(* PLC project Cell Example , CTH FIX1 1.0, author CTH SS2 *)
(* stored: companyURL www.chalmers.se, creationDateTime 2008-03-19 20:31:26, version 1.0, modificationDateTime 2008-04-03 16:58:09, organization SS2, language en-US *)

FUNCTION_BLOCK TwoPositionsMovement
  VAR_INPUT
    forward : BOOL := 0;
    backward : BOOL := 0;
    sensor_fwd : BOOL := 0;
    sensor_bwd : BOOL := 0;
  END_VAR
  VAR_OUTPUT
    in_forward : BOOL := 0;
    in_backward : BOOL := 0;
    out_forward : BOOL := 0;
    out_backward : BOOL := 0;
  END_VAR

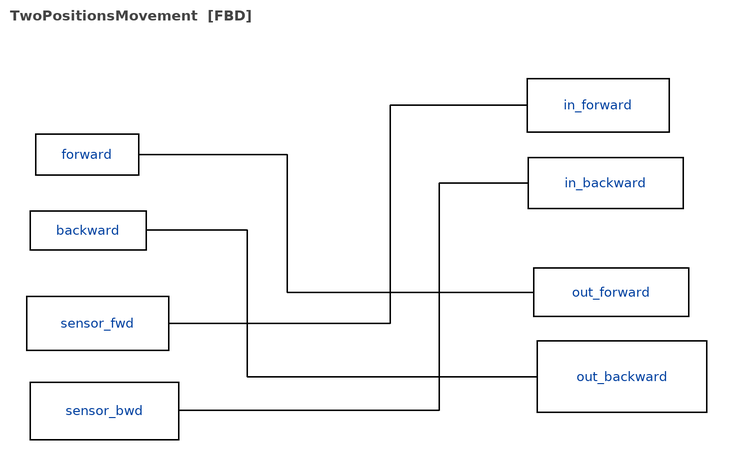
(* FBD diagram, written out as Structured Text *)
in_forward := sensor_fwd;
in_backward := sensor_bwd;
out_forward := forward;
out_backward := backward;
END_FUNCTION_BLOCK

FUNCTION_BLOCK PartDetection
  VAR_INPUT
    sensor_1 : BOOL := 0;
    sensor_2 : BOOL := 0;
  END_VAR
  VAR_OUTPUT
    part_present : BOOL := 0;
  END_VAR

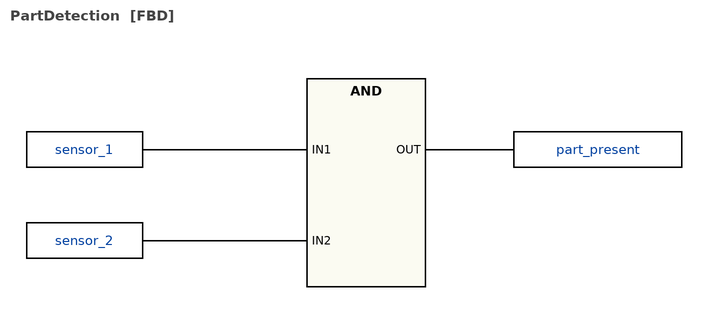
(* FBD diagram, written out as Structured Text *)
part_present := sensor_1 AND sensor_2;
END_FUNCTION_BLOCK

FUNCTION_BLOCK singleZoneBooking
  VAR_INPUT
    request_1 : BOOL := 0;
    request_2 : BOOL := 0;
  END_VAR
  VAR_OUTPUT
    booked_by_1 : BOOL := 0;
    booked_by_2 : BOOL := 0;
  END_VAR

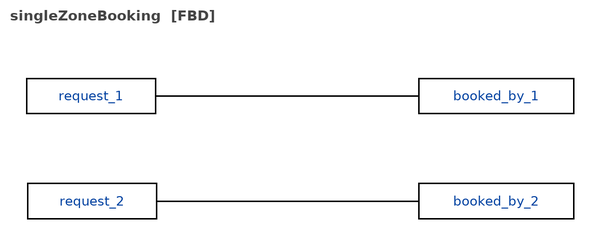
(* FBD diagram, written out as Structured Text *)
booked_by_1 := request_1;
booked_by_2 := request_2;
END_FUNCTION_BLOCK

PROGRAM EOP30
  VAR_EXTERNAL
    Op30_start : BOOL;
    positioning_in_home_pos : BOOL;
    fixation_in_locked : BOOL;
    clamp_in_open : BOOL;
    part_detection_part_present : BOOL;
    Op30_end : BOOL;
  END_VAR
  VAR  (* added by the conversion: wires and edge detectors of the diagram *)
    _AND8_OUT : BOOL;
  END_VAR

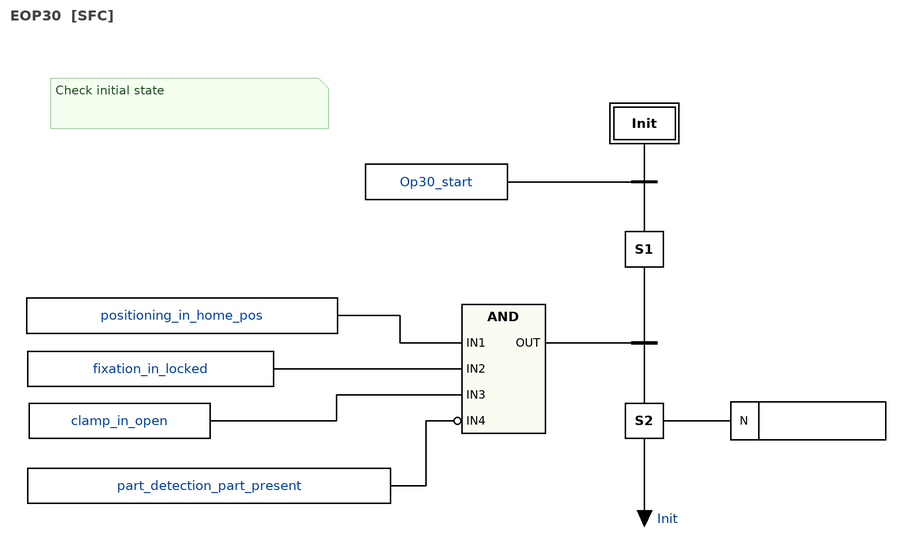
(* Check initial state *)
INITIAL_STEP Init:
  COMPUTE_FUNCTION_BLOCKS(S);
END_STEP
TRANSITION FROM Init TO S1
  := Op30_start;
END_TRANSITION
STEP S1:
END_STEP
TRANSITION FROM S1 TO S2
  := _AND8_OUT;
END_TRANSITION
STEP S2:
  S2_INLINE1(N, Op30_end);
END_STEP
ACTION S2_INLINE1:
END_ACTION
ACTION COMPUTE_FUNCTION_BLOCKS:  (* blocks drawn on the SFC sheet *)
  _AND8_OUT := positioning_in_home_pos AND fixation_in_locked AND clamp_in_open AND NOT part_detection_part_present;
END_ACTION
END_PROGRAM

PROGRAM EOP33
  VAR_EXTERNAL
    Op33_start : BOOL;
    Op33_end : BOOL;
    positioning_in_home_pos : BOOL;
    positioning_in_work_pos : BOOL;
    positioning_to_work_pos : BOOL;
    fixation_in_locked : BOOL;
    fixation_in_unlocked : BOOL;
    fixation_to_locked : BOOL;
    fixation_to_unlocked : BOOL;
    clamp_in_close : BOOL;
    part_detection_part_present : BOOL;
    Fix1_zone2_booked : BOOL;
    Fix1_zone3_booked : BOOL;
    Fix1_book_zone2 : BOOL;
    Fix1_book_zone3 : BOOL;
  END_VAR
  VAR  (* added by the conversion: wires and edge detectors of the diagram *)
    _AND7_OUT : BOOL;
    _AND15_OUT : BOOL;
    _AND27_OUT : BOOL;
    _AND38_OUT : BOOL;
  END_VAR

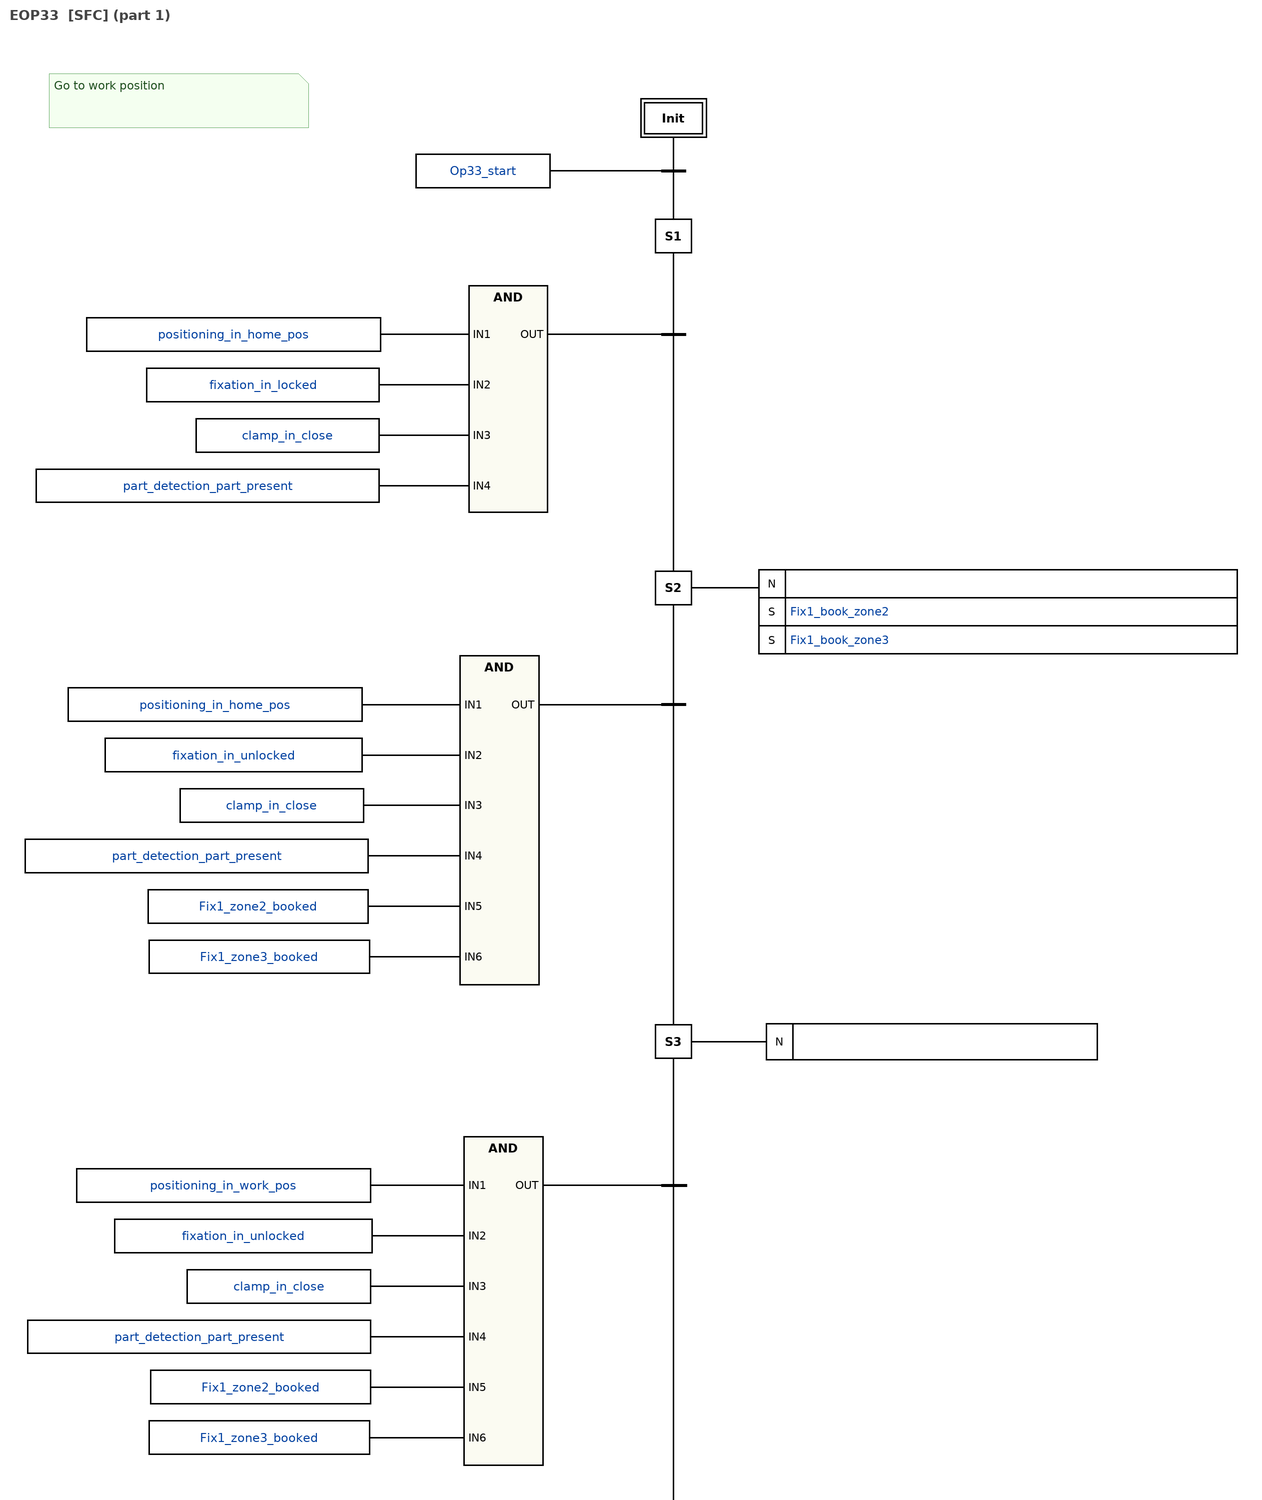
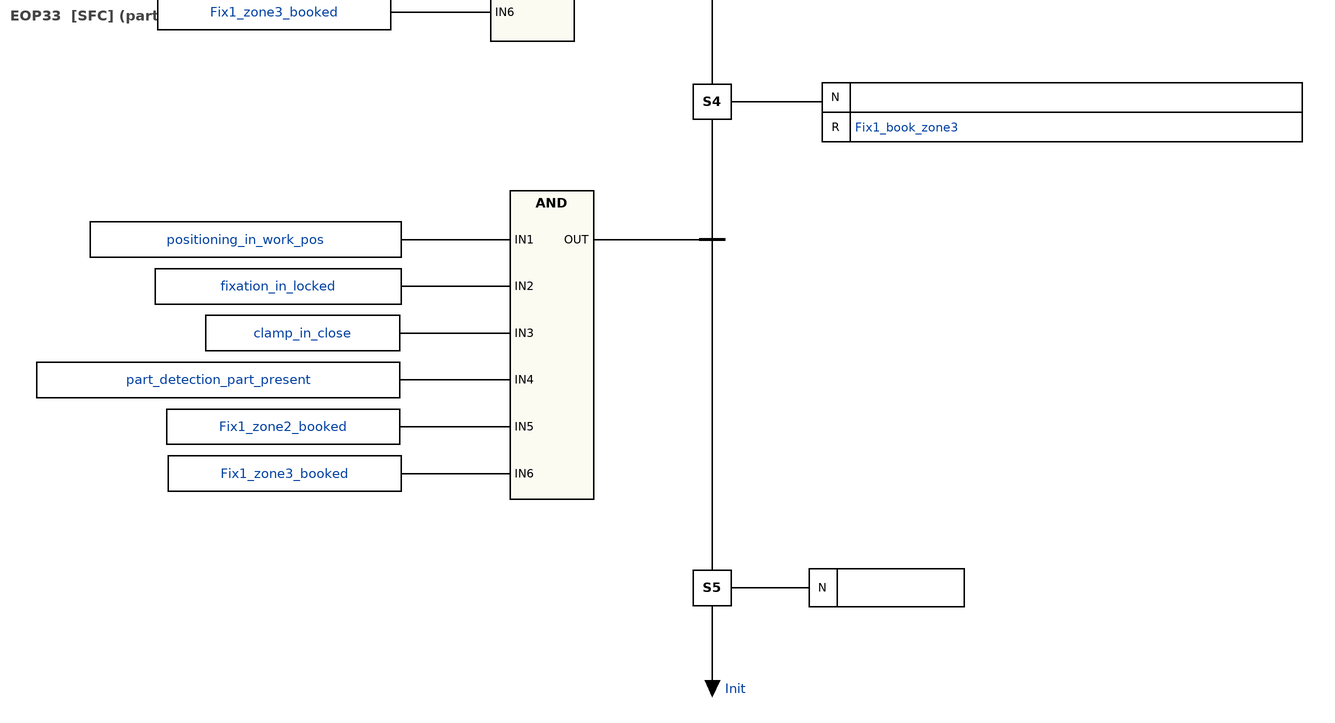
(* Go to work position *)
INITIAL_STEP Init:
  COMPUTE_FUNCTION_BLOCKS(S);
END_STEP
TRANSITION FROM Init TO S1
  := Op33_start;
END_TRANSITION
STEP S1:
END_STEP
TRANSITION FROM S1 TO S2
  := _AND7_OUT;
END_TRANSITION
STEP S2:
  S2_INLINE1(N, fixation_to_unlocked);
  Fix1_book_zone2(S);
  Fix1_book_zone3(S);
END_STEP
ACTION S2_INLINE1:
END_ACTION
TRANSITION FROM S2 TO S3
  := _AND15_OUT;
END_TRANSITION
STEP S3:
  S3_INLINE2(N, positioning_to_work_pos);
END_STEP
ACTION S3_INLINE2:
END_ACTION
TRANSITION FROM S3 TO S4
  := _AND27_OUT;
END_TRANSITION
STEP S4:
  S4_INLINE3(N, fixation_to_locked);
  Fix1_book_zone3(R);
END_STEP
ACTION S4_INLINE3:
END_ACTION
TRANSITION FROM S4 TO S5
  := _AND38_OUT;
END_TRANSITION
STEP S5:
  S5_INLINE4(N, Op33_end);
END_STEP
ACTION S5_INLINE4:
END_ACTION
ACTION COMPUTE_FUNCTION_BLOCKS:  (* blocks drawn on the SFC sheet *)
  _AND7_OUT := positioning_in_home_pos AND fixation_in_locked AND clamp_in_close AND part_detection_part_present;
  _AND15_OUT := positioning_in_home_pos AND fixation_in_unlocked AND clamp_in_close AND part_detection_part_present AND Fix1_zone2_booked AND Fix1_zone3_booked;
  _AND27_OUT := positioning_in_work_pos AND fixation_in_unlocked AND clamp_in_close AND part_detection_part_present AND Fix1_zone2_booked AND Fix1_zone3_booked;
  _AND38_OUT := positioning_in_work_pos AND fixation_in_locked AND clamp_in_close AND part_detection_part_present AND Fix1_zone2_booked AND Fix1_zone3_booked;
END_ACTION
END_PROGRAM

PROGRAM FunctionBlocks
  VAR_EXTERNAL
    positioning_in_home_pos : BOOL;
    positioning_to_home_pos : BOOL;
    positioning_output_to_home_pos : BOOL;
    positioning_sensor_in_home_pos : BOOL;
    positioning_in_work_pos : BOOL;
    positioning_to_work_pos : BOOL;
    positioning_output_to_work_pos : BOOL;
    positioning_sensor_in_work_pos : BOOL;
    fixation_in_locked : BOOL;
    fixation_to_locked : BOOL;
    fixation_output_to_locked : BOOL;
    fixation_sensor_in_locked : BOOL;
    fixation_in_unlocked : BOOL;
    fixation_to_unlocked : BOOL;
    fixation_output_to_unlocked : BOOL;
    fixation_sensor_in_unlocked : BOOL;
    clamp_in_open : BOOL;
    clamp_to_open : BOOL;
    clamp_output_to_open : BOOL;
    clamp_sensor_in_open : BOOL;
    clamp_in_close : BOOL;
    clamp_to_closed : BOOL;
    clamp_output_to_closed : BOOL;
    clamp_sensor_in_closed : BOOL;
    part_detection_part_present : BOOL;
    part_detection_sensor_1 : BOOL;
    part_detection_sensor_2 : BOOL;
    Fix1_book_zone2 : BOOL;
    Fix1_book_zone3 : BOOL;
    Fix1_zone2_booked : BOOL;
    Fix1_zone3_booked : BOOL;
  END_VAR
  VAR
    Positioning_1 : TwoPositionsMovement;
    PartDetection_1 : PartDetection;
    Fixation : TwoPositionsMovement;
    Clamp : TwoPositionsMovement;
    Zone2 : singleZoneBooking;
    Zone3 : singleZoneBooking;
  END_VAR

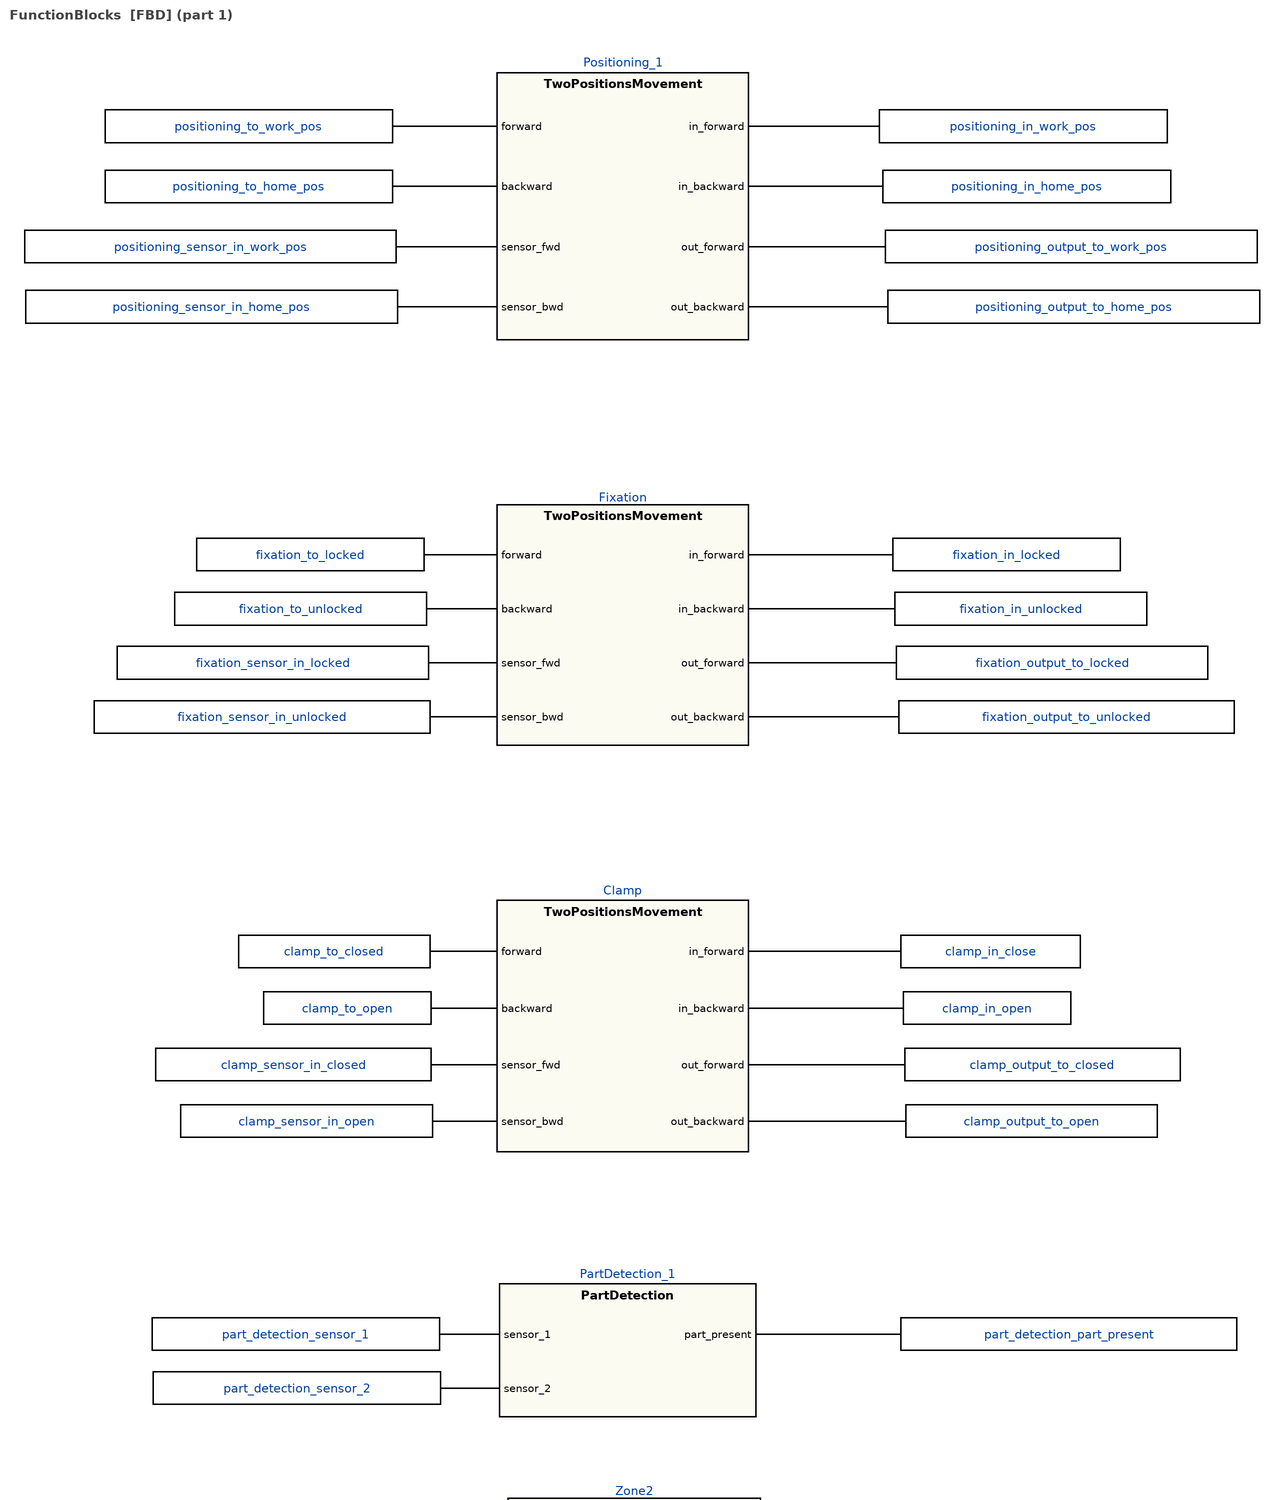
(* FBD diagram, written out as Structured Text *)
Positioning_1(forward := positioning_to_work_pos, backward := positioning_to_home_pos, sensor_fwd := positioning_sensor_in_work_pos, sensor_bwd := positioning_sensor_in_home_pos);
positioning_in_work_pos := Positioning_1.in_forward;
positioning_in_home_pos := Positioning_1.in_backward;
positioning_output_to_work_pos := Positioning_1.out_forward;
positioning_output_to_home_pos := Positioning_1.out_backward;
Fixation(forward := fixation_to_locked, backward := fixation_to_unlocked, sensor_fwd := fixation_sensor_in_locked, sensor_bwd := fixation_sensor_in_unlocked);
fixation_in_locked := Fixation.in_forward;
fixation_in_unlocked := Fixation.in_backward;
fixation_output_to_locked := Fixation.out_forward;
fixation_output_to_unlocked := Fixation.out_backward;
Clamp(forward := clamp_to_closed, backward := clamp_to_open, sensor_fwd := clamp_sensor_in_closed, sensor_bwd := clamp_sensor_in_open);
clamp_in_close := Clamp.in_forward;
clamp_in_open := Clamp.in_backward;
clamp_output_to_closed := Clamp.out_forward;
clamp_output_to_open := Clamp.out_backward;
PartDetection_1(sensor_1 := part_detection_sensor_1, sensor_2 := part_detection_sensor_2);
part_detection_part_present := PartDetection_1.part_present;
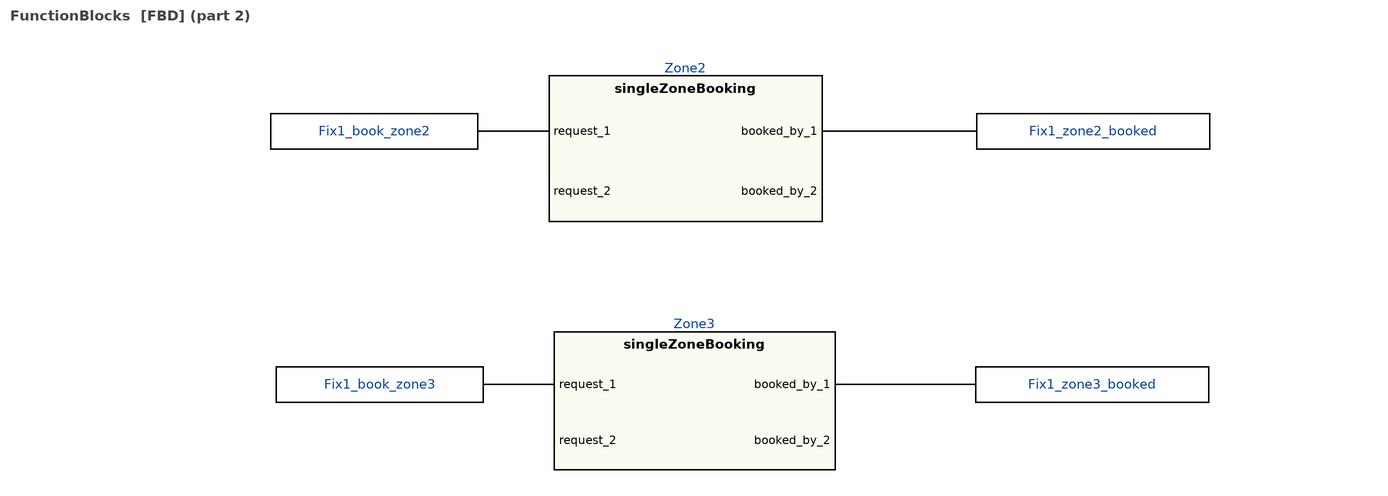
Zone2(request_1 := Fix1_book_zone2);
Fix1_zone2_booked := Zone2.booked_by_1;
Zone3(request_1 := Fix1_book_zone3);
Fix1_zone3_booked := Zone3.booked_by_1;
END_PROGRAM

PROGRAM COP1
  VAR_EXTERNAL
    Op30_start : BOOL;
    Op30_end : BOOL;
    Op31_start : BOOL;
    Op31_end : BOOL;
    Op32_start : BOOL;
    Op32_end : BOOL;
    Op33_start : BOOL;
    Op33_end : BOOL;
    Op34_start : BOOL;
    Op34_end : BOOL;
    Cop1_start : BOOL;
  END_VAR

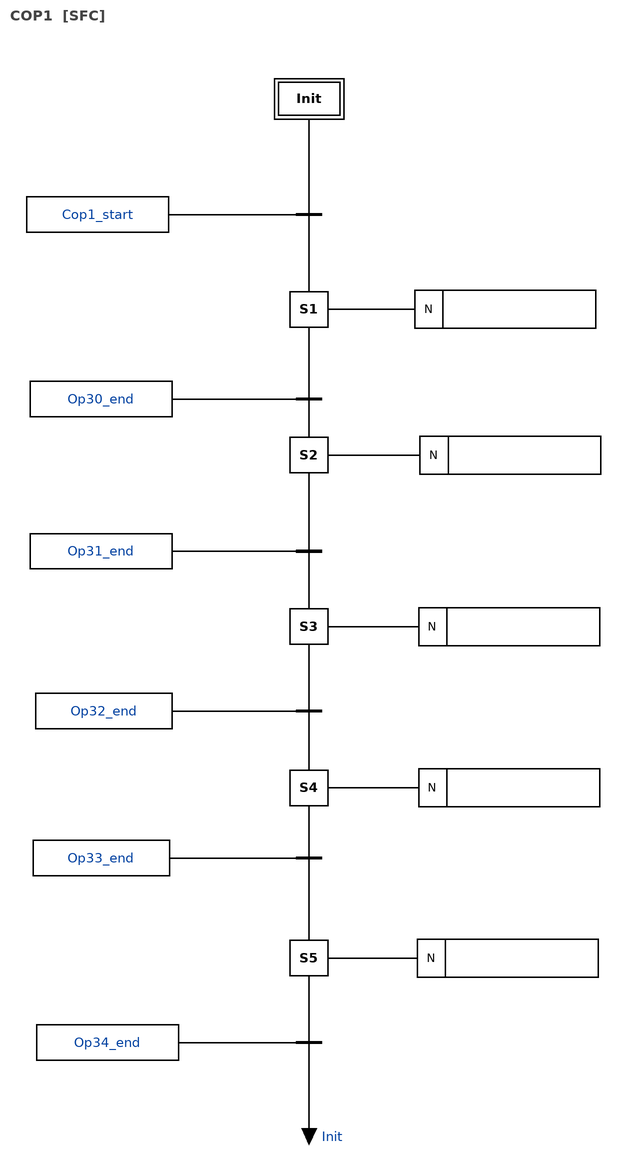
INITIAL_STEP Init:
END_STEP
TRANSITION FROM Init TO S1
  := Cop1_start;
END_TRANSITION
STEP S1:
  S1_INLINE1(N, Op30_start);
END_STEP
ACTION S1_INLINE1:
END_ACTION
TRANSITION FROM S1 TO S2
  := Op30_end;
END_TRANSITION
STEP S2:
  S2_INLINE2(N, Op31_start);
END_STEP
ACTION S2_INLINE2:
END_ACTION
TRANSITION FROM S2 TO S3
  := Op31_end;
END_TRANSITION
STEP S3:
  S3_INLINE3(N, Op32_start);
END_STEP
ACTION S3_INLINE3:
END_ACTION
TRANSITION FROM S3 TO S4
  := Op32_end;
END_TRANSITION
STEP S4:
  S4_INLINE4(N, Op33_start);
END_STEP
ACTION S4_INLINE4:
END_ACTION
TRANSITION FROM S4 TO S5
  := Op33_end;
END_TRANSITION
STEP S5:
  S5_INLINE5(N, Op34_start);
END_STEP
ACTION S5_INLINE5:
END_ACTION
TRANSITION FROM S5 TO Init
  := Op34_end;
END_TRANSITION
END_PROGRAM

CONFIGURATION ExampleCell
  VAR_GLOBAL
    Cop1_start : BOOL := 0;
    Cop1_end : BOOL := 0;
    Fix1_zone2_booked : BOOL := 0;
    Fix1_zone3_booked : BOOL := 0;
  END_VAR
  RESOURCE FIX1 ON PLC
    VAR_GLOBAL
      Op30_start : BOOL := 0;
      Op30_end : BOOL := 0;
      Op31_start : BOOL := 0;
      Op31_end : BOOL := 0;
      Op32_start : BOOL := 0;
      Op32_end : BOOL := 0;
      Op33_start : BOOL := 0;
      Op33_end : BOOL := 0;
      Op34_start : BOOL := 0;
      Op34_end : BOOL := 0;
      positioning_in_home_pos : BOOL := 0;
      positioning_to_home_pos : BOOL := 0;
      positioning_output_to_home_pos : BOOL := 0;
      positioning_sensor_in_home_pos : BOOL := 0;
      positioning_in_work_pos : BOOL := 0;
      positioning_to_work_pos : BOOL := 0;
      positioning_output_to_work_pos : BOOL := 0;
      positioning_sensor_in_work_pos : BOOL := 0;
      fixation_in_locked : BOOL := 0;
      fixation_to_locked : BOOL := 0;
      fixation_output_to_locked : BOOL := 0;
      fixation_sensor_in_locked : BOOL := 0;
      fixation_in_unlocked : BOOL := 0;
      fixation_to_unlocked : BOOL := 0;
      fixation_output_to_unlocked : BOOL := 0;
      fixation_sensor_in_unlocked : BOOL := 0;
      clamp_in_open : BOOL := 0;
      clamp_to_open : BOOL := 0;
      clamp_output_to_open : BOOL := 0;
      clamp_sensor_in_open : BOOL := 0;
      clamp_in_close : BOOL := 0;
      clamp_to_closed : BOOL := 0;
      clamp_output_to_closed : BOOL := 0;
      clamp_sensor_in_closed : BOOL := 0;
      part_detection_part_present : BOOL := 0;
      part_detection_sensor_1 : BOOL := 0;
      part_detection_sensor_2 : BOOL := 0;
      Fix1_book_zone2 : BOOL := 0;
      Fix1_book_zone3 : BOOL := 0;
    END_VAR
    TASK Task_COP1(SINGLE := Cop1_start, PRIORITY := 0);
    PROGRAM Instance_EOP30 WITH Task_COP1 : EOP30;
    PROGRAM Instance_EOP33 WITH Task_COP1 : EOP33;
    PROGRAM Instance_COP1 WITH Task_COP1 : COP1;
    PROGRAM Instance_FunctionBlocks WITH Task_COP1 : FunctionBlocks;
  END_RESOURCE
  RESOURCE COP2 ON PLC
  END_RESOURCE
END_CONFIGURATION
